FUNCTION_BLOCK FB_FlipTubeHandler EXTENDS FB_MzTool
VAR_INPUT
END_VAR
VAR_OUTPUT
END_VAR

SUPER^();	//FB_MzTool aufrufen

aObjProcData[nNotifyId] := stProcessData;

ACTION A_Reset:
//Ist noch eine Aktion aktiv?
IF nStateA_ResetSpec = 0 THEN 
	nStateA_ResetSpec := 80;
END_IF

SUPER^.A_Reset();
END_ACTION

METHOD FB_init : BOOL
VAR_INPUT
	bInitRetains : BOOL; // if TRUE, the retain variables are initialized (warm start / cold start)
	bInCopyCode : BOOL;  // if TRUE, the instance afterwards gets moved into the copy code (online change)
END_VAR
eObjectType := E_ObjectType.OBJECTTYPE_FlipTubeHandler;
eObjectGroup := E_ObjectGroup.OBJECTGROUP_MzTool OR E_ObjectGroup.OBJECTGROUP_Device;
END_METHOD

METHOD M_AddChild : ERRORID
VAR_INPUT
	pObject : POINTER TO FB_Object;
	nSlotNr	: UINT;
	nIndex 	: INT;
END_VAR
//Der Fliptube-Handler kann nur einen Exposure aufnehmen
IF pObject > 0 AND_THEN pObject^.P_eObjectType = E_ObjectType.OBJECTTYPE_Exposure THEN
	M_AddChild := SUPER^.M_AddChild(pObject,nSlotNr,nIndex);
ELSE
	M_AddChild := E_ErrorIdObjMgmt.ERRORID_InvalidParentObject;
END_IF
END_METHOD

METHOD M_CheckAction : ERRORID
VAR_INPUT
	refActionData 	: REFERENCE TO ST_ActionData;
	pCorrelObject	: POINTER TO FB_Object;
END_VAR
IF refActionData.eAction <> E_Action.ACTION_OpenCloseFlipTube THEN
	M_CheckAction := SUPER^.M_CheckAction(refActionData, pCorrelObject);
END_IF
END_METHOD

END_FUNCTION_BLOCK

(* stored: Version 1.1.0.1, ProductVersion 3.1.4024.5
   POU FB_FlipTubeHandler: Id {d3effa7c-5a8f-4a00-810f-8303acc03ac3}, SpecialFunc None
   Action A_Reset: Id {689d2207-57bf-495d-aa62-025be66a6ef0}
   Method FB_init: Id {8cf58970-be39-47bd-8243-37cf12a301a3}
   Method M_AddChild: Id {7323c4e1-b1d8-4a5b-a779-baa0aef5760e}
   Method M_CheckAction: Id {07491d0e-8398-4ae6-b62a-2b5bf418ed4e} *)
